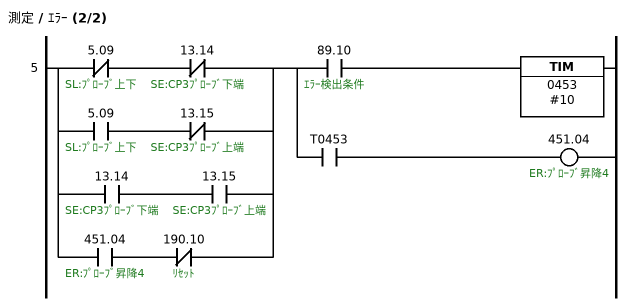
; rung 5
LDNOT 5.09  ; SL:ﾌﾟﾛｰﾌﾞ上下
ANDNOT 13.14  ; SE:CP3ﾌﾟﾛｰﾌﾞ下端
LD 5.09  ; SL:ﾌﾟﾛｰﾌﾞ上下
ANDNOT 13.15  ; SE:CP3ﾌﾟﾛｰﾌﾞ上端
ORLD
LD 13.14  ; SE:CP3ﾌﾟﾛｰﾌﾞ下端
AND 13.15  ; SE:CP3ﾌﾟﾛｰﾌﾞ上端
ORLD
LD 451.04  ; ER:ﾌﾟﾛｰﾌﾞ昇降4
ANDNOT 190.10  ; ﾘｾｯﾄ
ORLD
OUT TR0
AND 89.10  ; ｴﾗｰ検出条件
TIM 0453 #10
LD TR0
AND T0453
OUT 451.04  ; ER:ﾌﾟﾛｰﾌﾞ昇降4

### Section END
; rung 0
END(001)

## Program OV_RV (cyclic task 5)

### Section 制御

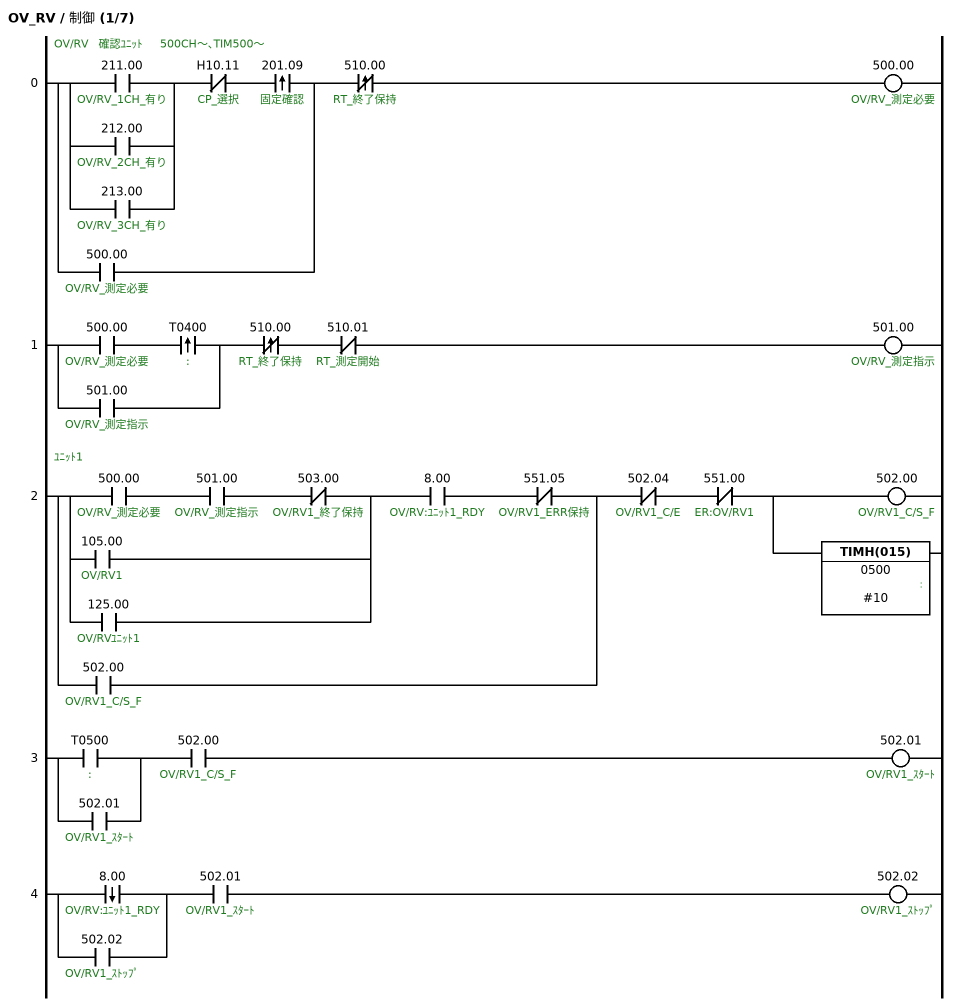
; rung 0: OV/RV   確認ﾕﾆｯﾄ     500CH～､TIM500～
LD 211.00  ; OV/RV_1CH_有り
OR 212.00  ; OV/RV_2CH_有り
OR 213.00  ; OV/RV_3CH_有り
ANDNOT H10.11  ; CP_選択
@AND 201.09  ; 固定確認
OR 500.00  ; OV/RV_測定必要
@ANDNOT 510.00  ; RT_終了保持
OUT 500.00  ; OV/RV_測定必要
; rung 1
LD 500.00  ; OV/RV_測定必要
@AND T0400  ; :
OR 501.00  ; OV/RV_測定指示
@ANDNOT 510.00  ; RT_終了保持
ANDNOT 510.01  ; RT_測定開始
OUT 501.00  ; OV/RV_測定指示
; rung 2: ﾕﾆｯﾄ1
LD 500.00  ; OV/RV_測定必要
AND 501.00  ; OV/RV_測定指示
ANDNOT 503.00  ; OV/RV1_終了保持
OR 105.00  ; OV/RV1
OR 125.00  ; OV/RVﾕﾆｯﾄ1
AND 8.00  ; OV/RV:ﾕﾆｯﾄ1_RDY
ANDNOT 551.05  ; OV/RV1_ERR保持
OR 502.00  ; OV/RV1_C/S_F
ANDNOT 502.04  ; OV/RV1_C/E
ANDNOT 551.00  ; ER:OV/RV1
OUT 502.00  ; OV/RV1_C/S_F
TIMH(015) 0500 #10  ; :
; rung 3
LD T0500  ; :
OR 502.01  ; OV/RV1_ｽﾀｰﾄ
AND 502.00  ; OV/RV1_C/S_F
OUT 502.01  ; OV/RV1_ｽﾀｰﾄ
; rung 4
%LD 8.00  ; OV/RV:ﾕﾆｯﾄ1_RDY
OR 502.02  ; OV/RV1_ｽﾄｯﾌﾟ
AND 502.01  ; OV/RV1_ｽﾀｰﾄ
OUT 502.02  ; OV/RV1_ｽﾄｯﾌﾟ

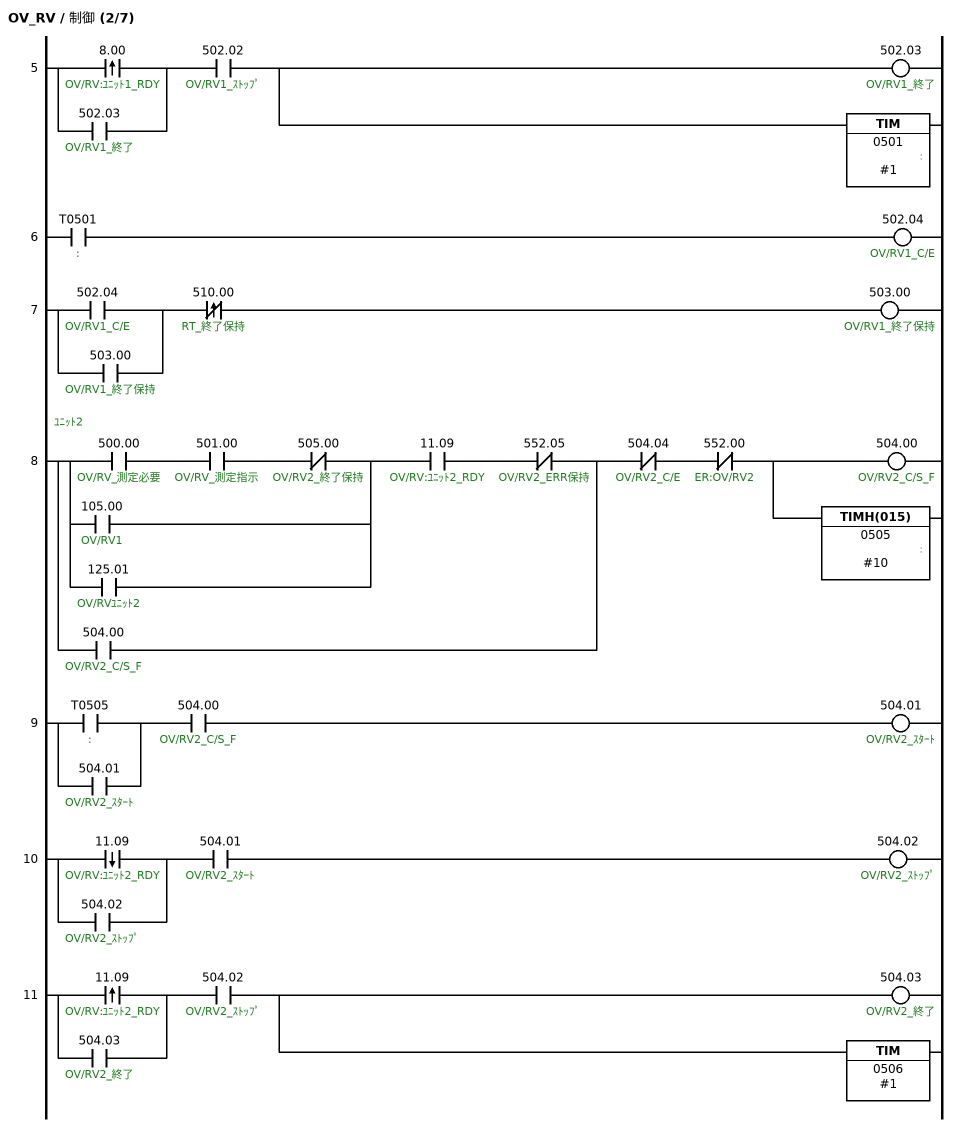
; rung 5
@LD 8.00  ; OV/RV:ﾕﾆｯﾄ1_RDY
OR 502.03  ; OV/RV1_終了
AND 502.02  ; OV/RV1_ｽﾄｯﾌﾟ
OUT 502.03  ; OV/RV1_終了
TIM 0501 #1  ; :
; rung 6
LD T0501  ; :
OUT 502.04  ; OV/RV1_C/E
; rung 7
LD 502.04  ; OV/RV1_C/E
OR 503.00  ; OV/RV1_終了保持
@ANDNOT 510.00  ; RT_終了保持
OUT 503.00  ; OV/RV1_終了保持
; rung 8: ﾕﾆｯﾄ2
LD 500.00  ; OV/RV_測定必要
AND 501.00  ; OV/RV_測定指示
ANDNOT 505.00  ; OV/RV2_終了保持
OR 105.00  ; OV/RV1
OR 125.01  ; OV/RVﾕﾆｯﾄ2
AND 11.09  ; OV/RV:ﾕﾆｯﾄ2_RDY
ANDNOT 552.05  ; OV/RV2_ERR保持
OR 504.00  ; OV/RV2_C/S_F
ANDNOT 504.04  ; OV/RV2_C/E
ANDNOT 552.00  ; ER:OV/RV2
OUT 504.00  ; OV/RV2_C/S_F
TIMH(015) 0505 #10  ; :
; rung 9
LD T0505  ; :
OR 504.01  ; OV/RV2_ｽﾀｰﾄ
AND 504.00  ; OV/RV2_C/S_F
OUT 504.01  ; OV/RV2_ｽﾀｰﾄ
; rung 10
%LD 11.09  ; OV/RV:ﾕﾆｯﾄ2_RDY
OR 504.02  ; OV/RV2_ｽﾄｯﾌﾟ
AND 504.01  ; OV/RV2_ｽﾀｰﾄ
OUT 504.02  ; OV/RV2_ｽﾄｯﾌﾟ
; rung 11
@LD 11.09  ; OV/RV:ﾕﾆｯﾄ2_RDY
OR 504.03  ; OV/RV2_終了
AND 504.02  ; OV/RV2_ｽﾄｯﾌﾟ
OUT 504.03  ; OV/RV2_終了
TIM 0506 #1

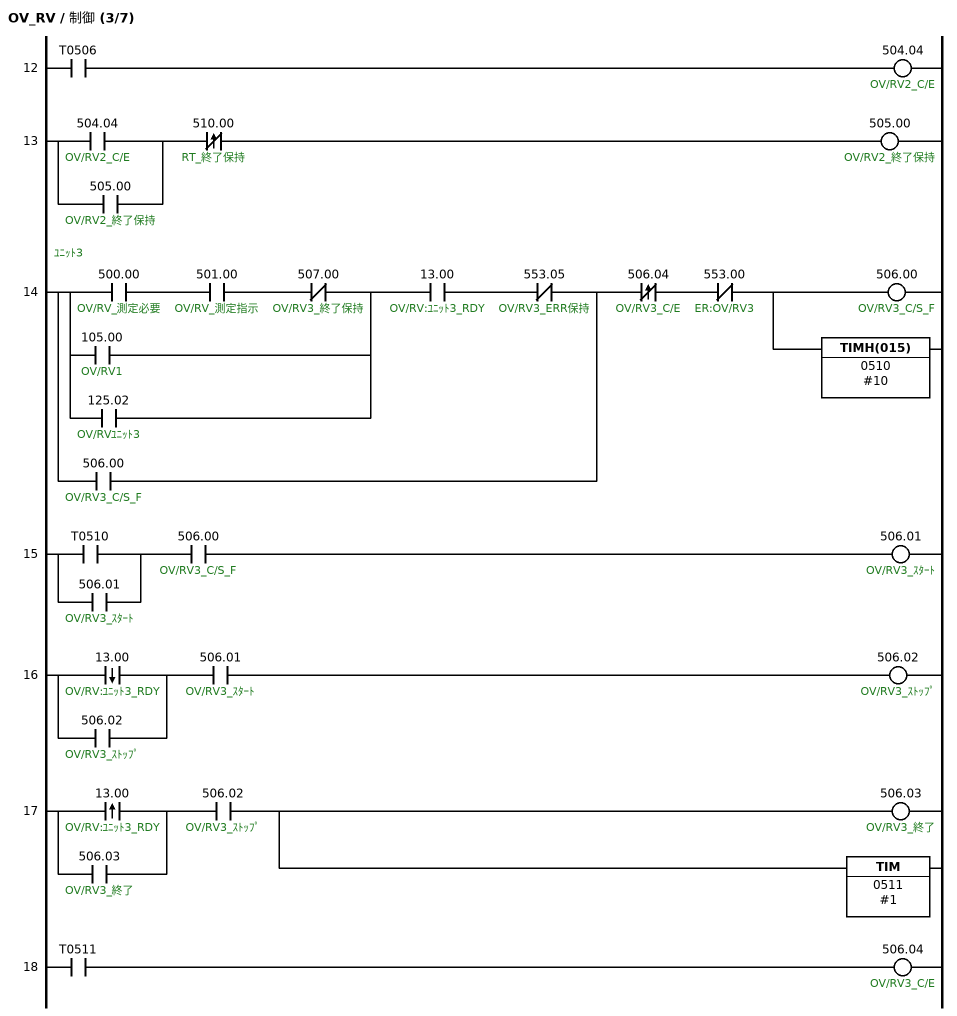
; rung 12
LD T0506
OUT 504.04  ; OV/RV2_C/E
; rung 13
LD 504.04  ; OV/RV2_C/E
OR 505.00  ; OV/RV2_終了保持
@ANDNOT 510.00  ; RT_終了保持
OUT 505.00  ; OV/RV2_終了保持
; rung 14: ﾕﾆｯﾄ3
LD 500.00  ; OV/RV_測定必要
AND 501.00  ; OV/RV_測定指示
ANDNOT 507.00  ; OV/RV3_終了保持
OR 105.00  ; OV/RV1
OR 125.02  ; OV/RVﾕﾆｯﾄ3
AND 13.00  ; OV/RV:ﾕﾆｯﾄ3_RDY
ANDNOT 553.05  ; OV/RV3_ERR保持
OR 506.00  ; OV/RV3_C/S_F
@ANDNOT 506.04  ; OV/RV3_C/E
ANDNOT 553.00  ; ER:OV/RV3
OUT 506.00  ; OV/RV3_C/S_F
TIMH(015) 0510 #10
; rung 15
LD T0510
OR 506.01  ; OV/RV3_ｽﾀｰﾄ
AND 506.00  ; OV/RV3_C/S_F
OUT 506.01  ; OV/RV3_ｽﾀｰﾄ
; rung 16
%LD 13.00  ; OV/RV:ﾕﾆｯﾄ3_RDY
OR 506.02  ; OV/RV3_ｽﾄｯﾌﾟ
AND 506.01  ; OV/RV3_ｽﾀｰﾄ
OUT 506.02  ; OV/RV3_ｽﾄｯﾌﾟ
; rung 17
@LD 13.00  ; OV/RV:ﾕﾆｯﾄ3_RDY
OR 506.03  ; OV/RV3_終了
AND 506.02  ; OV/RV3_ｽﾄｯﾌﾟ
OUT 506.03  ; OV/RV3_終了
TIM 0511 #1
; rung 18
LD T0511
OUT 506.04  ; OV/RV3_C/E

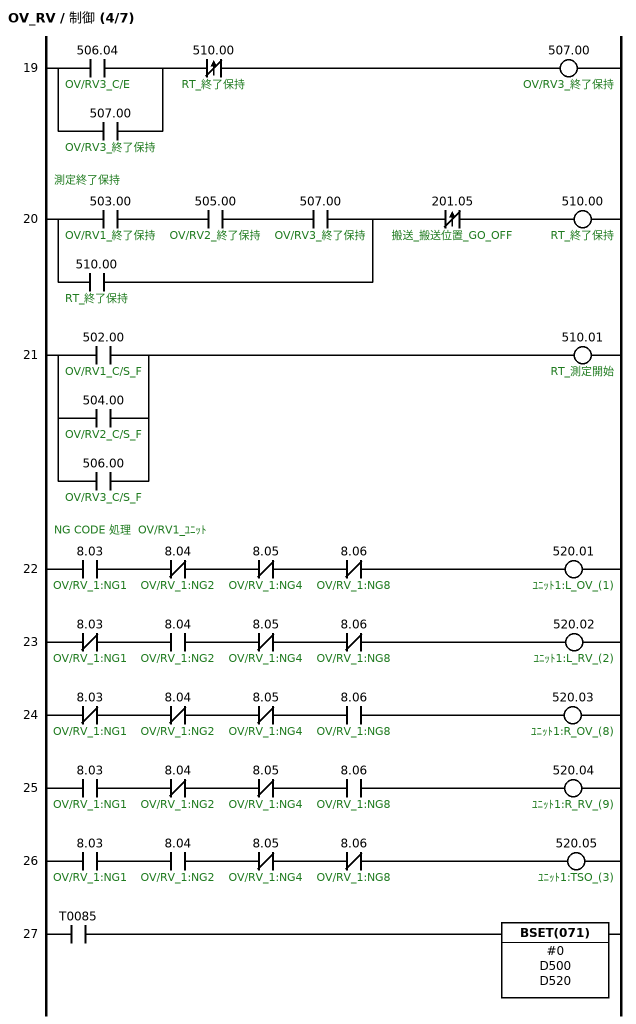
; rung 19
LD 506.04  ; OV/RV3_C/E
OR 507.00  ; OV/RV3_終了保持
@ANDNOT 510.00  ; RT_終了保持
OUT 507.00  ; OV/RV3_終了保持
; rung 20: 測定終了保持
LD 503.00  ; OV/RV1_終了保持
AND 505.00  ; OV/RV2_終了保持
AND 507.00  ; OV/RV3_終了保持
OR 510.00  ; RT_終了保持
@ANDNOT 201.05  ; 搬送_搬送位置_GO_OFF
OUT 510.00  ; RT_終了保持
; rung 21
LD 502.00  ; OV/RV1_C/S_F
OR 504.00  ; OV/RV2_C/S_F
OR 506.00  ; OV/RV3_C/S_F
OUT 510.01  ; RT_測定開始
; rung 22: NG CODE 処理  OV/RV1_ﾕﾆｯﾄ
LD 8.03  ; OV/RV_1:NG1
ANDNOT 8.04  ; OV/RV_1:NG2
ANDNOT 8.05  ; OV/RV_1:NG4
ANDNOT 8.06  ; OV/RV_1:NG8
OUT 520.01  ; ﾕﾆｯﾄ1:L_OV_(1)
; rung 23
LDNOT 8.03  ; OV/RV_1:NG1
AND 8.04  ; OV/RV_1:NG2
ANDNOT 8.05  ; OV/RV_1:NG4
ANDNOT 8.06  ; OV/RV_1:NG8
OUT 520.02  ; ﾕﾆｯﾄ1:L_RV_(2)
; rung 24
LDNOT 8.03  ; OV/RV_1:NG1
ANDNOT 8.04  ; OV/RV_1:NG2
ANDNOT 8.05  ; OV/RV_1:NG4
AND 8.06  ; OV/RV_1:NG8
OUT 520.03  ; ﾕﾆｯﾄ1:R_OV_(8)
; rung 25
LD 8.03  ; OV/RV_1:NG1
ANDNOT 8.04  ; OV/RV_1:NG2
ANDNOT 8.05  ; OV/RV_1:NG4
AND 8.06  ; OV/RV_1:NG8
OUT 520.04  ; ﾕﾆｯﾄ1:R_RV_(9)
; rung 26
LD 8.03  ; OV/RV_1:NG1
AND 8.04  ; OV/RV_1:NG2
ANDNOT 8.05  ; OV/RV_1:NG4
ANDNOT 8.06  ; OV/RV_1:NG8
OUT 520.05  ; ﾕﾆｯﾄ1:TSO_(3)
; rung 27
LD T0085
BSET(071) #0 D500 D520

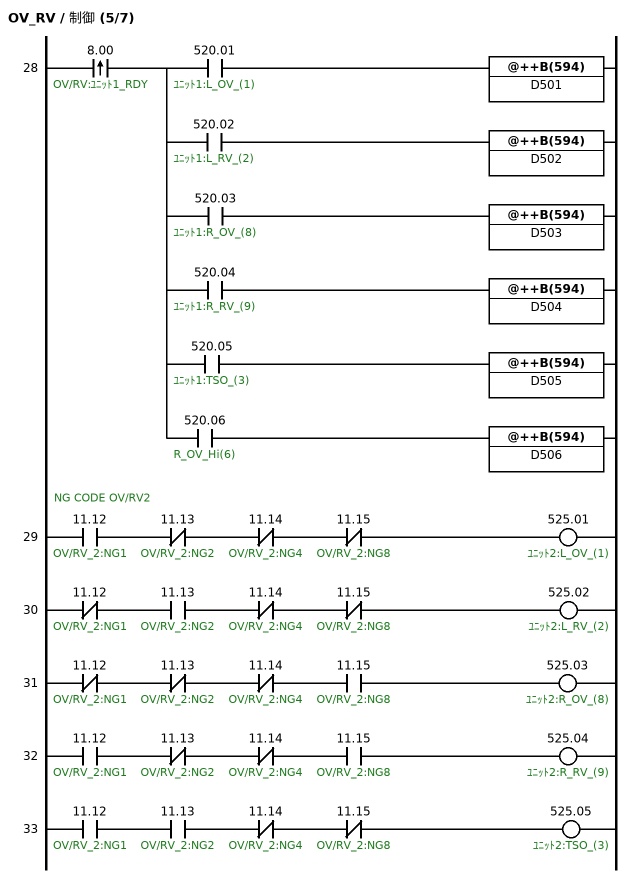
; rung 28
@LD 8.00  ; OV/RV:ﾕﾆｯﾄ1_RDY
OUT TR0
AND 520.01  ; ﾕﾆｯﾄ1:L_OV_(1)
@++B(594) D501
LD TR0
AND 520.02  ; ﾕﾆｯﾄ1:L_RV_(2)
@++B(594) D502
LD TR0
AND 520.03  ; ﾕﾆｯﾄ1:R_OV_(8)
@++B(594) D503
LD TR0
AND 520.04  ; ﾕﾆｯﾄ1:R_RV_(9)
@++B(594) D504
LD TR0
AND 520.05  ; ﾕﾆｯﾄ1:TSO_(3)
@++B(594) D505
LD TR0
AND 520.06  ; R_OV_Hi(6)
@++B(594) D506
; rung 29: NG CODE OV/RV2
LD 11.12  ; OV/RV_2:NG1
ANDNOT 11.13  ; OV/RV_2:NG2
ANDNOT 11.14  ; OV/RV_2:NG4
ANDNOT 11.15  ; OV/RV_2:NG8
OUT 525.01  ; ﾕﾆｯﾄ2:L_OV_(1)
; rung 30
LDNOT 11.12  ; OV/RV_2:NG1
AND 11.13  ; OV/RV_2:NG2
ANDNOT 11.14  ; OV/RV_2:NG4
ANDNOT 11.15  ; OV/RV_2:NG8
OUT 525.02  ; ﾕﾆｯﾄ2:L_RV_(2)
; rung 31
LDNOT 11.12  ; OV/RV_2:NG1
ANDNOT 11.13  ; OV/RV_2:NG2
ANDNOT 11.14  ; OV/RV_2:NG4
AND 11.15  ; OV/RV_2:NG8
OUT 525.03  ; ﾕﾆｯﾄ2:R_OV_(8)
; rung 32
LD 11.12  ; OV/RV_2:NG1
ANDNOT 11.13  ; OV/RV_2:NG2
ANDNOT 11.14  ; OV/RV_2:NG4
AND 11.15  ; OV/RV_2:NG8
OUT 525.04  ; ﾕﾆｯﾄ2:R_RV_(9)
; rung 33
LD 11.12  ; OV/RV_2:NG1
AND 11.13  ; OV/RV_2:NG2
ANDNOT 11.14  ; OV/RV_2:NG4
ANDNOT 11.15  ; OV/RV_2:NG8
OUT 525.05  ; ﾕﾆｯﾄ2:TSO_(3)

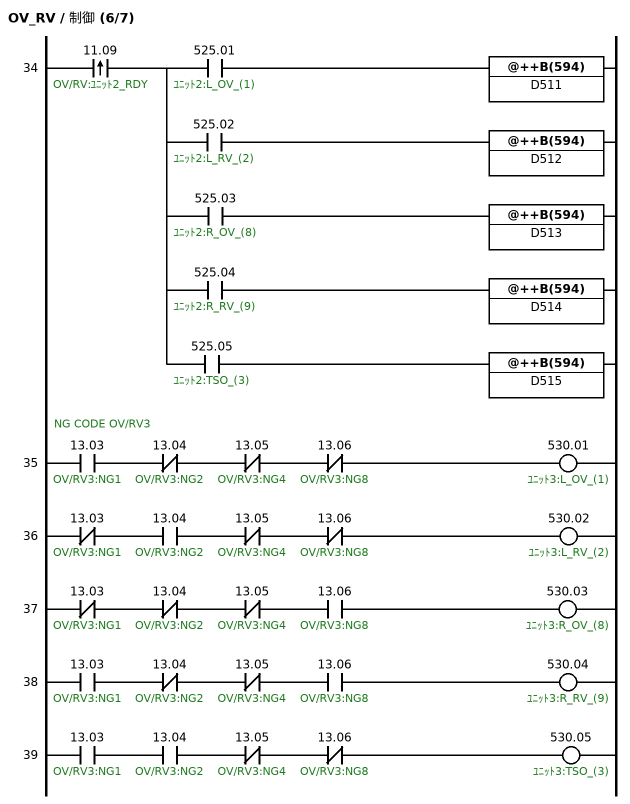
; rung 34
@LD 11.09  ; OV/RV:ﾕﾆｯﾄ2_RDY
OUT TR0
AND 525.01  ; ﾕﾆｯﾄ2:L_OV_(1)
@++B(594) D511
LD TR0
AND 525.02  ; ﾕﾆｯﾄ2:L_RV_(2)
@++B(594) D512
LD TR0
AND 525.03  ; ﾕﾆｯﾄ2:R_OV_(8)
@++B(594) D513
LD TR0
AND 525.04  ; ﾕﾆｯﾄ2:R_RV_(9)
@++B(594) D514
LD TR0
AND 525.05  ; ﾕﾆｯﾄ2:TSO_(3)
@++B(594) D515
; rung 35: NG CODE OV/RV3
LD 13.03  ; OV/RV3:NG1
ANDNOT 13.04  ; OV/RV3:NG2
ANDNOT 13.05  ; OV/RV3:NG4
ANDNOT 13.06  ; OV/RV3:NG8
OUT 530.01  ; ﾕﾆｯﾄ3:L_OV_(1)
; rung 36
LDNOT 13.03  ; OV/RV3:NG1
AND 13.04  ; OV/RV3:NG2
ANDNOT 13.05  ; OV/RV3:NG4
ANDNOT 13.06  ; OV/RV3:NG8
OUT 530.02  ; ﾕﾆｯﾄ3:L_RV_(2)
; rung 37
LDNOT 13.03  ; OV/RV3:NG1
ANDNOT 13.04  ; OV/RV3:NG2
ANDNOT 13.05  ; OV/RV3:NG4
AND 13.06  ; OV/RV3:NG8
OUT 530.03  ; ﾕﾆｯﾄ3:R_OV_(8)
; rung 38
LD 13.03  ; OV/RV3:NG1
ANDNOT 13.04  ; OV/RV3:NG2
ANDNOT 13.05  ; OV/RV3:NG4
AND 13.06  ; OV/RV3:NG8
OUT 530.04  ; ﾕﾆｯﾄ3:R_RV_(9)
; rung 39
LD 13.03  ; OV/RV3:NG1
AND 13.04  ; OV/RV3:NG2
ANDNOT 13.05  ; OV/RV3:NG4
ANDNOT 13.06  ; OV/RV3:NG8
OUT 530.05  ; ﾕﾆｯﾄ3:TSO_(3)

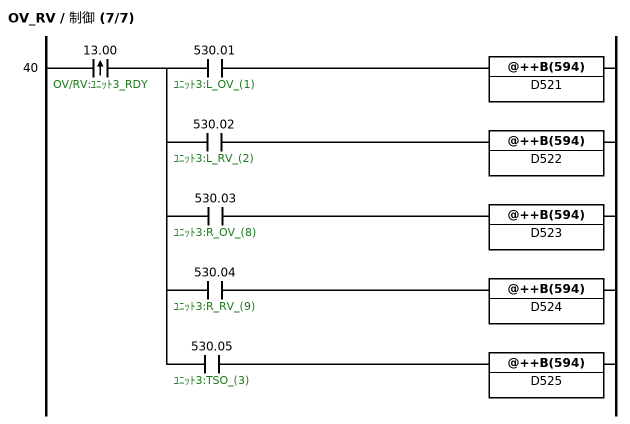
; rung 40
@LD 13.00  ; OV/RV:ﾕﾆｯﾄ3_RDY
OUT TR0
AND 530.01  ; ﾕﾆｯﾄ3:L_OV_(1)
@++B(594) D521
LD TR0
AND 530.02  ; ﾕﾆｯﾄ3:L_RV_(2)
@++B(594) D522
LD TR0
AND 530.03  ; ﾕﾆｯﾄ3:R_OV_(8)
@++B(594) D523
LD TR0
AND 530.04  ; ﾕﾆｯﾄ3:R_RV_(9)
@++B(594) D524
LD TR0
AND 530.05  ; ﾕﾆｯﾄ3:TSO_(3)
@++B(594) D525

### Section 出力
; rung 0: 出力

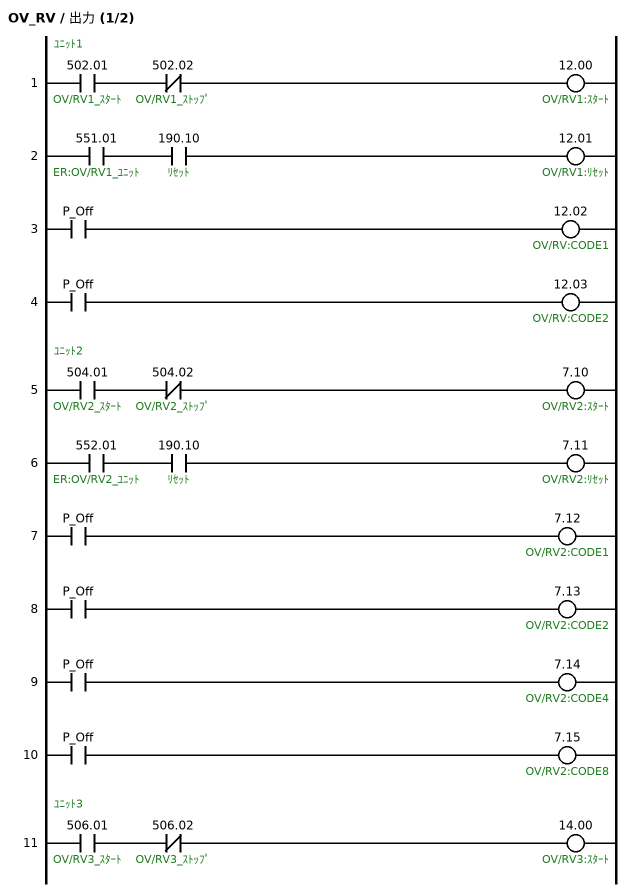
; rung 1: ﾕﾆｯﾄ1
LD 502.01  ; OV/RV1_ｽﾀｰﾄ
ANDNOT 502.02  ; OV/RV1_ｽﾄｯﾌﾟ
OUT 12.00  ; OV/RV1:ｽﾀｰﾄ
; rung 2
LD 551.01  ; ER:OV/RV1_ﾕﾆｯﾄ
AND 190.10  ; ﾘｾｯﾄ
OUT 12.01  ; OV/RV1:ﾘｾｯﾄ
; rung 3
LD P_Off
OUT 12.02  ; OV/RV:CODE1
; rung 4
LD P_Off
OUT 12.03  ; OV/RV:CODE2
; rung 5: ﾕﾆｯﾄ2
LD 504.01  ; OV/RV2_ｽﾀｰﾄ
ANDNOT 504.02  ; OV/RV2_ｽﾄｯﾌﾟ
OUT 7.10  ; OV/RV2:ｽﾀｰﾄ
; rung 6
LD 552.01  ; ER:OV/RV2_ﾕﾆｯﾄ
AND 190.10  ; ﾘｾｯﾄ
OUT 7.11  ; OV/RV2:ﾘｾｯﾄ
; rung 7
LD P_Off
OUT 7.12  ; OV/RV2:CODE1
; rung 8
LD P_Off
OUT 7.13  ; OV/RV2:CODE2
; rung 9
LD P_Off
OUT 7.14  ; OV/RV2:CODE4
; rung 10
LD P_Off
OUT 7.15  ; OV/RV2:CODE8
; rung 11: ﾕﾆｯﾄ3
LD 506.01  ; OV/RV3_ｽﾀｰﾄ
ANDNOT 506.02  ; OV/RV3_ｽﾄｯﾌﾟ
OUT 14.00  ; OV/RV3:ｽﾀｰﾄ

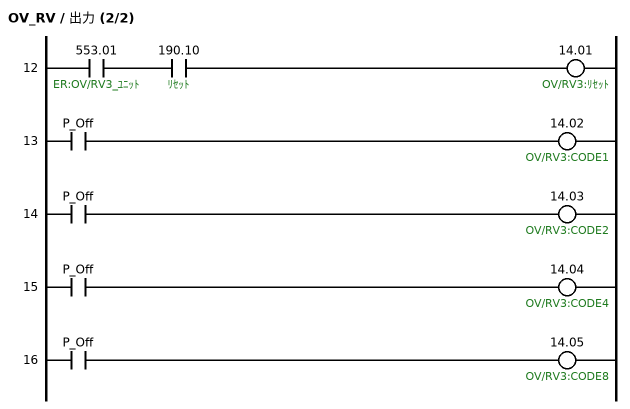
; rung 12
LD 553.01  ; ER:OV/RV3_ﾕﾆｯﾄ
AND 190.10  ; ﾘｾｯﾄ
OUT 14.01  ; OV/RV3:ﾘｾｯﾄ
; rung 13
LD P_Off
OUT 14.02  ; OV/RV3:CODE1
; rung 14
LD P_Off
OUT 14.03  ; OV/RV3:CODE2
; rung 15
LD P_Off
OUT 14.04  ; OV/RV3:CODE4
; rung 16
LD P_Off
OUT 14.05  ; OV/RV3:CODE8

### Section ｴﾗｰ

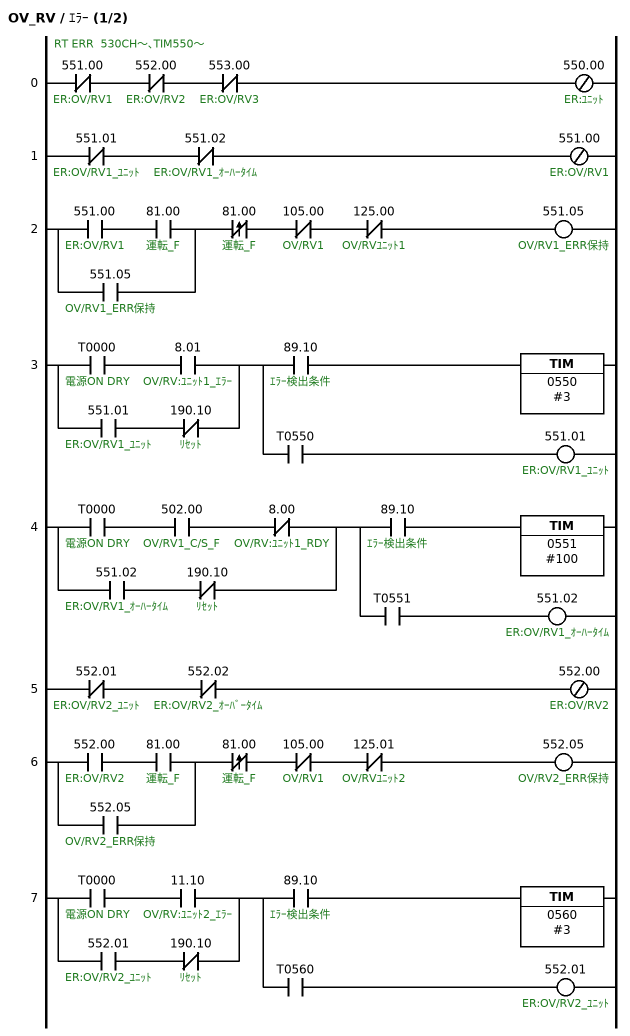
; rung 0: RT ERR  530CH～､TIM550～
LDNOT 551.00  ; ER:OV/RV1
ANDNOT 552.00  ; ER:OV/RV2
ANDNOT 553.00  ; ER:OV/RV3
OUTNOT 550.00  ; ER:ﾕﾆｯﾄ
; rung 1
LDNOT 551.01  ; ER:OV/RV1_ﾕﾆｯﾄ
ANDNOT 551.02  ; ER:OV/RV1_ｵｰﾊｰﾀｲﾑ
OUTNOT 551.00  ; ER:OV/RV1
; rung 2
LD 551.00  ; ER:OV/RV1
AND 81.00  ; 運転_F
OR 551.05  ; OV/RV1_ERR保持
@ANDNOT 81.00  ; 運転_F
ANDNOT 105.00  ; OV/RV1
ANDNOT 125.00  ; OV/RVﾕﾆｯﾄ1
OUT 551.05  ; OV/RV1_ERR保持
; rung 3
LD T0000  ; 電源ON DRY
AND 8.01  ; OV/RV:ﾕﾆｯﾄ1_ｴﾗｰ
LD 551.01  ; ER:OV/RV1_ﾕﾆｯﾄ
ANDNOT 190.10  ; ﾘｾｯﾄ
ORLD
OUT TR0
AND 89.10  ; ｴﾗｰ検出条件
TIM 0550 #3
LD TR0
AND T0550
OUT 551.01  ; ER:OV/RV1_ﾕﾆｯﾄ
; rung 4
LD T0000  ; 電源ON DRY
AND 502.00  ; OV/RV1_C/S_F
ANDNOT 8.00  ; OV/RV:ﾕﾆｯﾄ1_RDY
LD 551.02  ; ER:OV/RV1_ｵｰﾊｰﾀｲﾑ
ANDNOT 190.10  ; ﾘｾｯﾄ
ORLD
OUT TR0
AND 89.10  ; ｴﾗｰ検出条件
TIM 0551 #100
LD TR0
AND T0551
OUT 551.02  ; ER:OV/RV1_ｵｰﾊｰﾀｲﾑ
; rung 5
LDNOT 552.01  ; ER:OV/RV2_ﾕﾆｯﾄ
ANDNOT 552.02  ; ER:OV/RV2_ｵｰﾊﾞｰﾀｲﾑ
OUTNOT 552.00  ; ER:OV/RV2
; rung 6
LD 552.00  ; ER:OV/RV2
AND 81.00  ; 運転_F
OR 552.05  ; OV/RV2_ERR保持
@ANDNOT 81.00  ; 運転_F
ANDNOT 105.00  ; OV/RV1
ANDNOT 125.01  ; OV/RVﾕﾆｯﾄ2
OUT 552.05  ; OV/RV2_ERR保持
; rung 7
LD T0000  ; 電源ON DRY
AND 11.10  ; OV/RV:ﾕﾆｯﾄ2_ｴﾗｰ
LD 552.01  ; ER:OV/RV2_ﾕﾆｯﾄ
ANDNOT 190.10  ; ﾘｾｯﾄ
ORLD
OUT TR0
AND 89.10  ; ｴﾗｰ検出条件
TIM 0560 #3
LD TR0
AND T0560
OUT 552.01  ; ER:OV/RV2_ﾕﾆｯﾄ

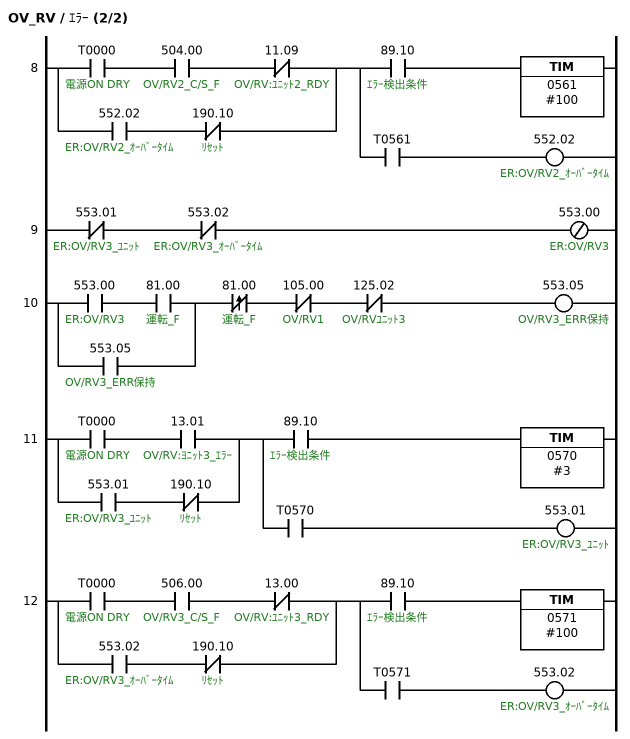
; rung 8
LD T0000  ; 電源ON DRY
AND 504.00  ; OV/RV2_C/S_F
ANDNOT 11.09  ; OV/RV:ﾕﾆｯﾄ2_RDY
LD 552.02  ; ER:OV/RV2_ｵｰﾊﾞｰﾀｲﾑ
ANDNOT 190.10  ; ﾘｾｯﾄ
ORLD
OUT TR0
AND 89.10  ; ｴﾗｰ検出条件
TIM 0561 #100
LD TR0
AND T0561
OUT 552.02  ; ER:OV/RV2_ｵｰﾊﾞｰﾀｲﾑ
; rung 9
LDNOT 553.01  ; ER:OV/RV3_ﾕﾆｯﾄ
ANDNOT 553.02  ; ER:OV/RV3_ｵｰﾊﾞｰﾀｲﾑ
OUTNOT 553.00  ; ER:OV/RV3
; rung 10
LD 553.00  ; ER:OV/RV3
AND 81.00  ; 運転_F
OR 553.05  ; OV/RV3_ERR保持
@ANDNOT 81.00  ; 運転_F
ANDNOT 105.00  ; OV/RV1
ANDNOT 125.02  ; OV/RVﾕﾆｯﾄ3
OUT 553.05  ; OV/RV3_ERR保持
; rung 11
LD T0000  ; 電源ON DRY
AND 13.01  ; OV/RV:ﾖﾆｯﾄ3_ｴﾗｰ
LD 553.01  ; ER:OV/RV3_ﾕﾆｯﾄ
ANDNOT 190.10  ; ﾘｾｯﾄ
ORLD
OUT TR0
AND 89.10  ; ｴﾗｰ検出条件
TIM 0570 #3
LD TR0
AND T0570
OUT 553.01  ; ER:OV/RV3_ﾕﾆｯﾄ
; rung 12
LD T0000  ; 電源ON DRY
AND 506.00  ; OV/RV3_C/S_F
ANDNOT 13.00  ; OV/RV:ﾕﾆｯﾄ3_RDY
LD 553.02  ; ER:OV/RV3_ｵｰﾊﾞｰﾀｲﾑ
ANDNOT 190.10  ; ﾘｾｯﾄ
ORLD
OUT TR0
AND 89.10  ; ｴﾗｰ検出条件
TIM 0571 #100
LD TR0
AND T0571
OUT 553.02  ; ER:OV/RV3_ｵｰﾊﾞｰﾀｲﾑ

### Section END
; rung 0
END(001)

## Program CP (cyclic task 6)

### Section 制御

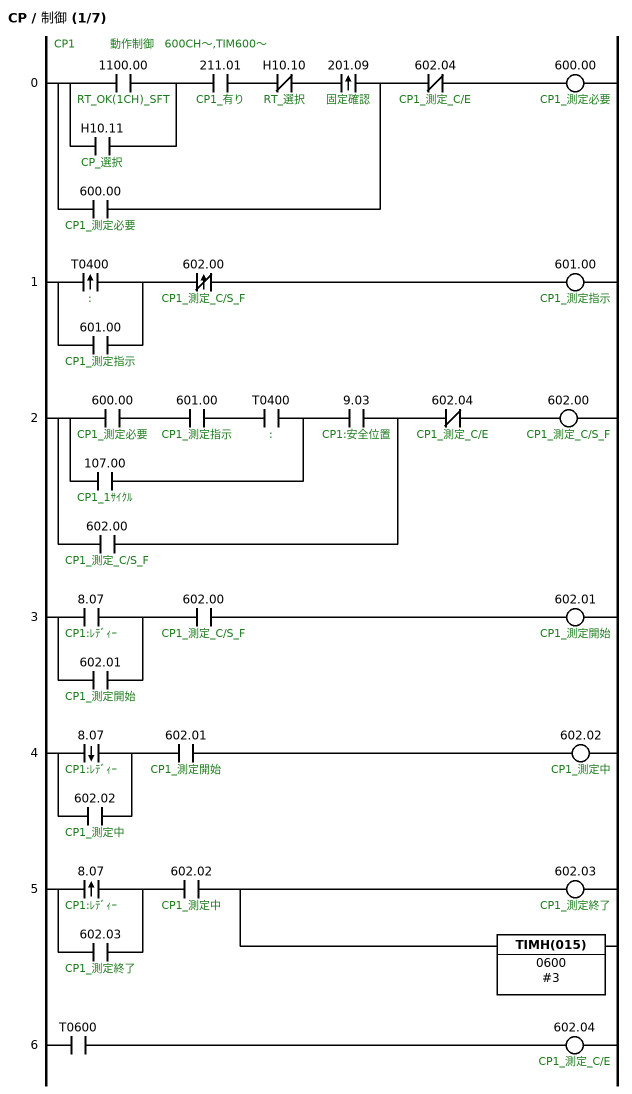
; rung 0: CP1          動作制御   600CH～,TIM600～
LD 1100.00  ; RT_OK(1CH)_SFT
OR H10.11  ; CP_選択
AND 211.01  ; CP1_有り
ANDNOT H10.10  ; RT_選択
@AND 201.09  ; 固定確認
OR 600.00  ; CP1_測定必要
ANDNOT 602.04  ; CP1_測定_C/E
OUT 600.00  ; CP1_測定必要
; rung 1
@LD T0400  ; :
OR 601.00  ; CP1_測定指示
@ANDNOT 602.00  ; CP1_測定_C/S_F
OUT 601.00  ; CP1_測定指示
; rung 2
LD 600.00  ; CP1_測定必要
AND 601.00  ; CP1_測定指示
AND T0400  ; :
OR 107.00  ; CP1_1ｻｲｸﾙ
AND 9.03  ; CP1:安全位置
OR 602.00  ; CP1_測定_C/S_F
ANDNOT 602.04  ; CP1_測定_C/E
OUT 602.00  ; CP1_測定_C/S_F
; rung 3
LD 8.07  ; CP1:ﾚﾃﾞｨｰ
OR 602.01  ; CP1_測定開始
AND 602.00  ; CP1_測定_C/S_F
OUT 602.01  ; CP1_測定開始
; rung 4
%LD 8.07  ; CP1:ﾚﾃﾞｨｰ
OR 602.02  ; CP1_測定中
AND 602.01  ; CP1_測定開始
OUT 602.02  ; CP1_測定中
; rung 5
@LD 8.07  ; CP1:ﾚﾃﾞｨｰ
OR 602.03  ; CP1_測定終了
AND 602.02  ; CP1_測定中
OUT 602.03  ; CP1_測定終了
TIMH(015) 0600 #3
; rung 6
LD T0600
OUT 602.04  ; CP1_測定_C/E

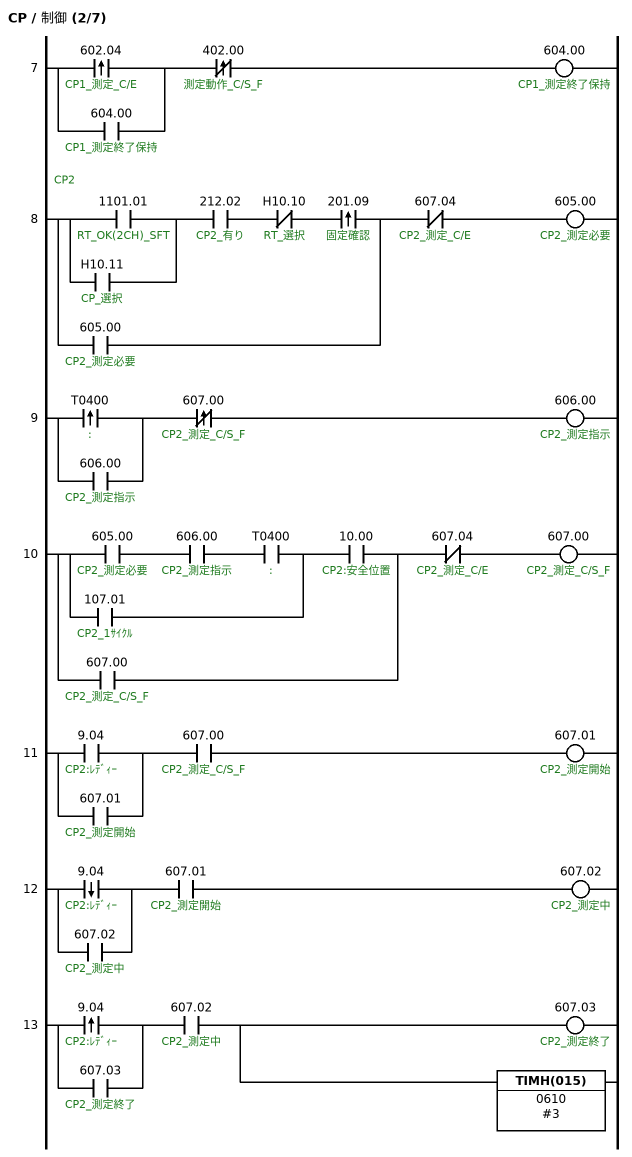
; rung 7
@LD 602.04  ; CP1_測定_C/E
OR 604.00  ; CP1_測定終了保持
@ANDNOT 402.00  ; 測定動作_C/S_F
OUT 604.00  ; CP1_測定終了保持
; rung 8: CP2
LD 1101.01  ; RT_OK(2CH)_SFT
OR H10.11  ; CP_選択
AND 212.02  ; CP2_有り
ANDNOT H10.10  ; RT_選択
@AND 201.09  ; 固定確認
OR 605.00  ; CP2_測定必要
ANDNOT 607.04  ; CP2_測定_C/E
OUT 605.00  ; CP2_測定必要
; rung 9
@LD T0400  ; :
OR 606.00  ; CP2_測定指示
@ANDNOT 607.00  ; CP2_測定_C/S_F
OUT 606.00  ; CP2_測定指示
; rung 10
LD 605.00  ; CP2_測定必要
AND 606.00  ; CP2_測定指示
AND T0400  ; :
OR 107.01  ; CP2_1ｻｲｸﾙ
AND 10.00  ; CP2:安全位置
OR 607.00  ; CP2_測定_C/S_F
ANDNOT 607.04  ; CP2_測定_C/E
OUT 607.00  ; CP2_測定_C/S_F
; rung 11
LD 9.04  ; CP2:ﾚﾃﾞｨｰ
OR 607.01  ; CP2_測定開始
AND 607.00  ; CP2_測定_C/S_F
OUT 607.01  ; CP2_測定開始
; rung 12
%LD 9.04  ; CP2:ﾚﾃﾞｨｰ
OR 607.02  ; CP2_測定中
AND 607.01  ; CP2_測定開始
OUT 607.02  ; CP2_測定中
; rung 13
@LD 9.04  ; CP2:ﾚﾃﾞｨｰ
OR 607.03  ; CP2_測定終了
AND 607.02  ; CP2_測定中
OUT 607.03  ; CP2_測定終了
TIMH(015) 0610 #3

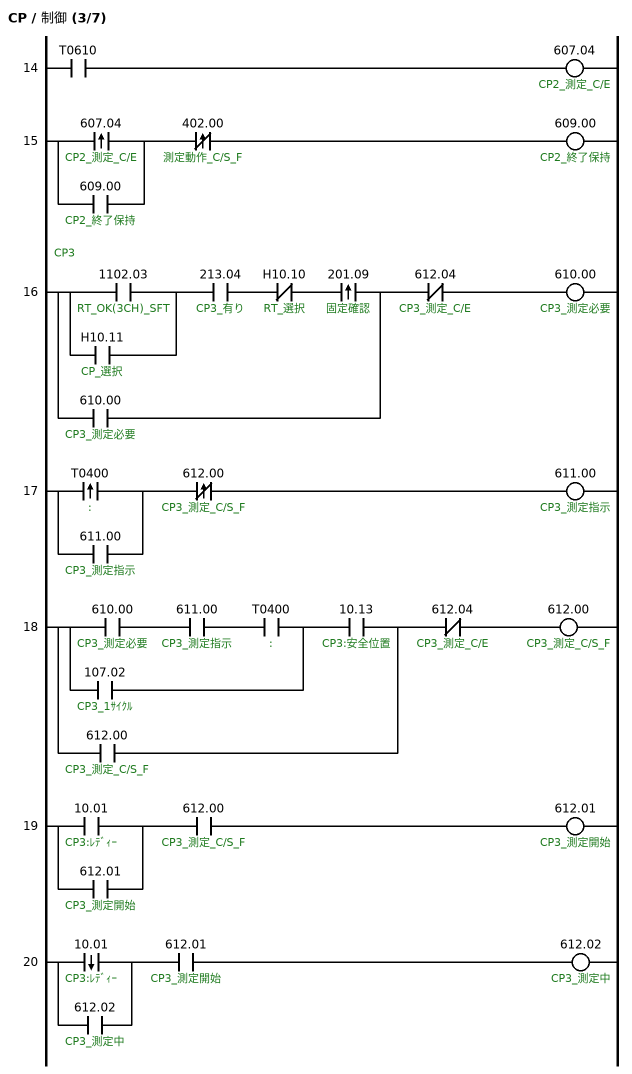
; rung 14
LD T0610
OUT 607.04  ; CP2_測定_C/E
; rung 15
@LD 607.04  ; CP2_測定_C/E
OR 609.00  ; CP2_終了保持
@ANDNOT 402.00  ; 測定動作_C/S_F
OUT 609.00  ; CP2_終了保持
; rung 16: CP3
LD 1102.03  ; RT_OK(3CH)_SFT
OR H10.11  ; CP_選択
AND 213.04  ; CP3_有り
ANDNOT H10.10  ; RT_選択
@AND 201.09  ; 固定確認
OR 610.00  ; CP3_測定必要
ANDNOT 612.04  ; CP3_測定_C/E
OUT 610.00  ; CP3_測定必要
; rung 17
@LD T0400  ; :
OR 611.00  ; CP3_測定指示
@ANDNOT 612.00  ; CP3_測定_C/S_F
OUT 611.00  ; CP3_測定指示
; rung 18
LD 610.00  ; CP3_測定必要
AND 611.00  ; CP3_測定指示
AND T0400  ; :
OR 107.02  ; CP3_1ｻｲｸﾙ
AND 10.13  ; CP3:安全位置
OR 612.00  ; CP3_測定_C/S_F
ANDNOT 612.04  ; CP3_測定_C/E
OUT 612.00  ; CP3_測定_C/S_F
; rung 19
LD 10.01  ; CP3:ﾚﾃﾞｨｰ
OR 612.01  ; CP3_測定開始
AND 612.00  ; CP3_測定_C/S_F
OUT 612.01  ; CP3_測定開始
; rung 20
%LD 10.01  ; CP3:ﾚﾃﾞｨｰ
OR 612.02  ; CP3_測定中
AND 612.01  ; CP3_測定開始
OUT 612.02  ; CP3_測定中

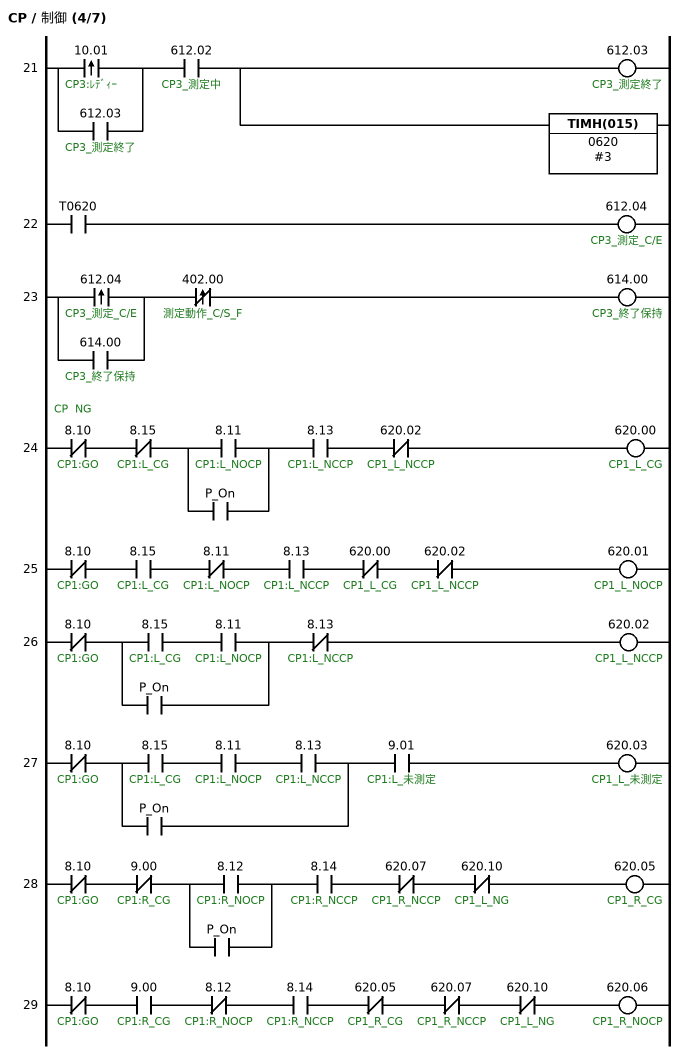
; rung 21
@LD 10.01  ; CP3:ﾚﾃﾞｨｰ
OR 612.03  ; CP3_測定終了
AND 612.02  ; CP3_測定中
OUT 612.03  ; CP3_測定終了
TIMH(015) 0620 #3
; rung 22
LD T0620
OUT 612.04  ; CP3_測定_C/E
; rung 23
@LD 612.04  ; CP3_測定_C/E
OR 614.00  ; CP3_終了保持
@ANDNOT 402.00  ; 測定動作_C/S_F
OUT 614.00  ; CP3_終了保持
; rung 24: CP  NG
LDNOT 8.10  ; CP1:GO
ANDNOT 8.15  ; CP1:L_CG
LD 8.11  ; CP1:L_NOCP
OR P_On  // 2015/11/13変更
ANDLD
AND 8.13  ; CP1:L_NCCP
ANDNOT 620.02  ; CP1_L_NCCP  // 2015/11/13変更
OUT 620.00  ; CP1_L_CG
; rung 25
LDNOT 8.10  ; CP1:GO
AND 8.15  ; CP1:L_CG
ANDNOT 8.11  ; CP1:L_NOCP
AND 8.13  ; CP1:L_NCCP
ANDNOT 620.00  ; CP1_L_CG
ANDNOT 620.02  ; CP1_L_NCCP  // 2015/11/13変更
OUT 620.01  ; CP1_L_NOCP
; rung 26
LDNOT 8.10  ; CP1:GO
LD 8.15  ; CP1:L_CG
AND 8.11  ; CP1:L_NOCP
OR P_On  // 2015/11/13変更
ANDLD
ANDNOT 8.13  ; CP1:L_NCCP
OUT 620.02  ; CP1_L_NCCP
; rung 27
LDNOT 8.10  ; CP1:GO
LD 8.15  ; CP1:L_CG
AND 8.11  ; CP1:L_NOCP
AND 8.13  ; CP1:L_NCCP
OR P_On  // 2015/11/13変更
ANDLD
AND 9.01  ; CP1:L_未測定  // 2015/11/13変更
OUT 620.03  ; CP1_L_未測定
; rung 28
LDNOT 8.10  ; CP1:GO
ANDNOT 9.00  ; CP1:R_CG
LD 8.12  ; CP1:R_NOCP
OR P_On  // 2015/11/13変更
ANDLD
AND 8.14  ; CP1:R_NCCP
ANDNOT 620.07  ; CP1_R_NCCP
ANDNOT 620.10  ; CP1_L_NG
OUT 620.05  ; CP1_R_CG
; rung 29
LDNOT 8.10  ; CP1:GO
AND 9.00  ; CP1:R_CG
ANDNOT 8.12  ; CP1:R_NOCP
AND 8.14  ; CP1:R_NCCP
ANDNOT 620.05  ; CP1_R_CG
ANDNOT 620.07  ; CP1_R_NCCP
ANDNOT 620.10  ; CP1_L_NG
OUT 620.06  ; CP1_R_NOCP

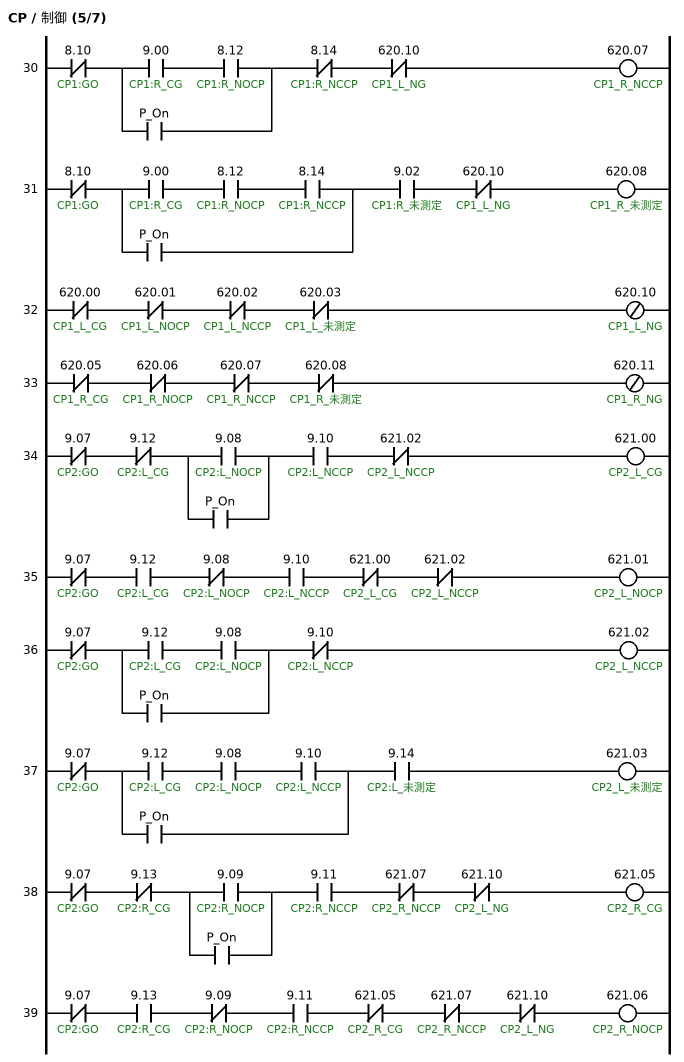
; rung 30
LDNOT 8.10  ; CP1:GO
LD 9.00  ; CP1:R_CG
AND 8.12  ; CP1:R_NOCP
OR P_On  // 2015/11/13変更
ANDLD
ANDNOT 8.14  ; CP1:R_NCCP
ANDNOT 620.10  ; CP1_L_NG
OUT 620.07  ; CP1_R_NCCP
; rung 31
LDNOT 8.10  ; CP1:GO
LD 9.00  ; CP1:R_CG
AND 8.12  ; CP1:R_NOCP
AND 8.14  ; CP1:R_NCCP
OR P_On  // 2015/11/13変更
ANDLD
AND 9.02  ; CP1:R_未測定  // 2015/11/13変更
ANDNOT 620.10  ; CP1_L_NG
OUT 620.08  ; CP1_R_未測定
; rung 32
LDNOT 620.00  ; CP1_L_CG
ANDNOT 620.01  ; CP1_L_NOCP
ANDNOT 620.02  ; CP1_L_NCCP
ANDNOT 620.03  ; CP1_L_未測定
OUTNOT 620.10  ; CP1_L_NG
; rung 33
LDNOT 620.05  ; CP1_R_CG
ANDNOT 620.06  ; CP1_R_NOCP
ANDNOT 620.07  ; CP1_R_NCCP
ANDNOT 620.08  ; CP1_R_未測定
OUTNOT 620.11  ; CP1_R_NG
; rung 34
LDNOT 9.07  ; CP2:GO
ANDNOT 9.12  ; CP2:L_CG
LD 9.08  ; CP2:L_NOCP
OR P_On  // 2015/11/13変更
ANDLD
AND 9.10  ; CP2:L_NCCP
ANDNOT 621.02  ; CP2_L_NCCP
OUT 621.00  ; CP2_L_CG
; rung 35
LDNOT 9.07  ; CP2:GO
AND 9.12  ; CP2:L_CG
ANDNOT 9.08  ; CP2:L_NOCP
AND 9.10  ; CP2:L_NCCP
ANDNOT 621.00  ; CP2_L_CG
ANDNOT 621.02  ; CP2_L_NCCP
OUT 621.01  ; CP2_L_NOCP
; rung 36
LDNOT 9.07  ; CP2:GO
LD 9.12  ; CP2:L_CG
AND 9.08  ; CP2:L_NOCP
OR P_On  // 2015/11/13変更
ANDLD
ANDNOT 9.10  ; CP2:L_NCCP
OUT 621.02  ; CP2_L_NCCP
; rung 37
LDNOT 9.07  ; CP2:GO
LD 9.12  ; CP2:L_CG
AND 9.08  ; CP2:L_NOCP
AND 9.10  ; CP2:L_NCCP
OR P_On  // 2015/11/13変更
ANDLD
AND 9.14  ; CP2:L_未測定  // 2015/11/13変更
OUT 621.03  ; CP2_L_未測定
; rung 38
LDNOT 9.07  ; CP2:GO
ANDNOT 9.13  ; CP2:R_CG
LD 9.09  ; CP2:R_NOCP
OR P_On  // 2015/11/13変更
ANDLD
AND 9.11  ; CP2:R_NCCP
ANDNOT 621.07  ; CP2_R_NCCP
ANDNOT 621.10  ; CP2_L_NG
OUT 621.05  ; CP2_R_CG
; rung 39
LDNOT 9.07  ; CP2:GO
AND 9.13  ; CP2:R_CG
ANDNOT 9.09  ; CP2:R_NOCP
AND 9.11  ; CP2:R_NCCP
ANDNOT 621.05  ; CP2_R_CG
ANDNOT 621.07  ; CP2_R_NCCP
ANDNOT 621.10  ; CP2_L_NG
OUT 621.06  ; CP2_R_NOCP

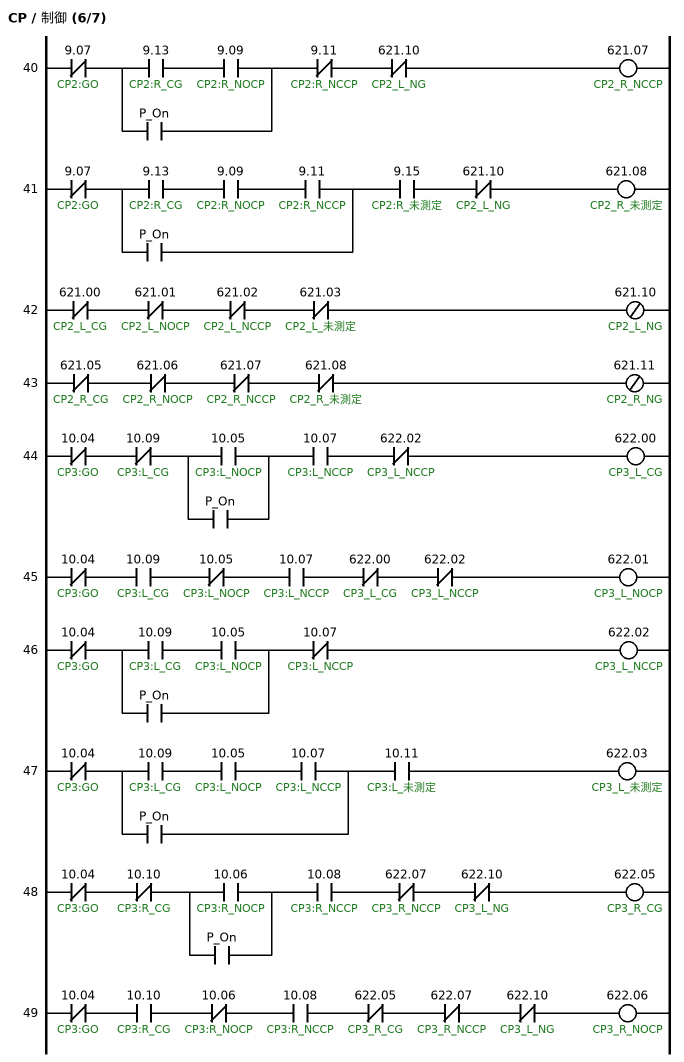
; rung 40
LDNOT 9.07  ; CP2:GO
LD 9.13  ; CP2:R_CG
AND 9.09  ; CP2:R_NOCP
OR P_On  // 2015/11/13変更
ANDLD
ANDNOT 9.11  ; CP2:R_NCCP
ANDNOT 621.10  ; CP2_L_NG
OUT 621.07  ; CP2_R_NCCP
; rung 41
LDNOT 9.07  ; CP2:GO
LD 9.13  ; CP2:R_CG
AND 9.09  ; CP2:R_NOCP
AND 9.11  ; CP2:R_NCCP
OR P_On  // 2015/11/13変更
ANDLD
AND 9.15  ; CP2:R_未測定  // 2015/11/13変更
ANDNOT 621.10  ; CP2_L_NG
OUT 621.08  ; CP2_R_未測定
; rung 42
LDNOT 621.00  ; CP2_L_CG
ANDNOT 621.01  ; CP2_L_NOCP
ANDNOT 621.02  ; CP2_L_NCCP
ANDNOT 621.03  ; CP2_L_未測定
OUTNOT 621.10  ; CP2_L_NG
; rung 43
LDNOT 621.05  ; CP2_R_CG
ANDNOT 621.06  ; CP2_R_NOCP
ANDNOT 621.07  ; CP2_R_NCCP
ANDNOT 621.08  ; CP2_R_未測定
OUTNOT 621.11  ; CP2_R_NG
; rung 44
LDNOT 10.04  ; CP3:GO
ANDNOT 10.09  ; CP3:L_CG
LD 10.05  ; CP3:L_NOCP
OR P_On  // 2015/11/13変更
ANDLD
AND 10.07  ; CP3:L_NCCP
ANDNOT 622.02  ; CP3_L_NCCP
OUT 622.00  ; CP3_L_CG
; rung 45
LDNOT 10.04  ; CP3:GO
AND 10.09  ; CP3:L_CG
ANDNOT 10.05  ; CP3:L_NOCP
AND 10.07  ; CP3:L_NCCP
ANDNOT 622.00  ; CP3_L_CG
ANDNOT 622.02  ; CP3_L_NCCP
OUT 622.01  ; CP3_L_NOCP
; rung 46
LDNOT 10.04  ; CP3:GO
LD 10.09  ; CP3:L_CG
AND 10.05  ; CP3:L_NOCP
OR P_On  // 2015/11/13変更
ANDLD
ANDNOT 10.07  ; CP3:L_NCCP
OUT 622.02  ; CP3_L_NCCP
; rung 47
LDNOT 10.04  ; CP3:GO
LD 10.09  ; CP3:L_CG
AND 10.05  ; CP3:L_NOCP
AND 10.07  ; CP3:L_NCCP
OR P_On  // 2015/11/13変更
ANDLD
AND 10.11  ; CP3:L_未測定  // 2015/11/13変更
OUT 622.03  ; CP3_L_未測定
; rung 48
LDNOT 10.04  ; CP3:GO
ANDNOT 10.10  ; CP3:R_CG
LD 10.06  ; CP3:R_NOCP
OR P_On  // 2015/11/13変更
ANDLD
AND 10.08  ; CP3:R_NCCP
ANDNOT 622.07  ; CP3_R_NCCP
ANDNOT 622.10  ; CP3_L_NG
OUT 622.05  ; CP3_R_CG
; rung 49
LDNOT 10.04  ; CP3:GO
AND 10.10  ; CP3:R_CG
ANDNOT 10.06  ; CP3:R_NOCP
AND 10.08  ; CP3:R_NCCP
ANDNOT 622.05  ; CP3_R_CG
ANDNOT 622.07  ; CP3_R_NCCP
ANDNOT 622.10  ; CP3_L_NG
OUT 622.06  ; CP3_R_NOCP

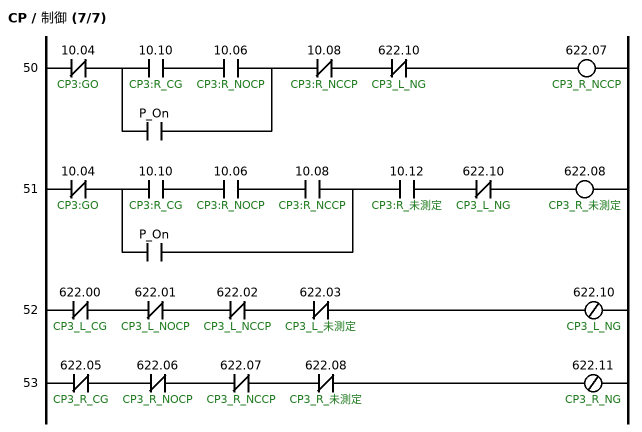
; rung 50
LDNOT 10.04  ; CP3:GO
LD 10.10  ; CP3:R_CG
AND 10.06  ; CP3:R_NOCP
OR P_On  // 2015/11/13変更
ANDLD
ANDNOT 10.08  ; CP3:R_NCCP
ANDNOT 622.10  ; CP3_L_NG
OUT 622.07  ; CP3_R_NCCP
; rung 51
LDNOT 10.04  ; CP3:GO
LD 10.10  ; CP3:R_CG
AND 10.06  ; CP3:R_NOCP
AND 10.08  ; CP3:R_NCCP
OR P_On  // 2015/11/13変更
ANDLD
AND 10.12  ; CP3:R_未測定  // 2015/11/13変更
ANDNOT 622.10  ; CP3_L_NG
OUT 622.08  ; CP3_R_未測定
; rung 52
LDNOT 622.00  ; CP3_L_CG
ANDNOT 622.01  ; CP3_L_NOCP
ANDNOT 622.02  ; CP3_L_NCCP
ANDNOT 622.03  ; CP3_L_未測定
OUTNOT 622.10  ; CP3_L_NG
; rung 53
LDNOT 622.05  ; CP3_R_CG
ANDNOT 622.06  ; CP3_R_NOCP
ANDNOT 622.07  ; CP3_R_NCCP
ANDNOT 622.08  ; CP3_R_未測定
OUTNOT 622.11  ; CP3_R_NG

### Section 出力

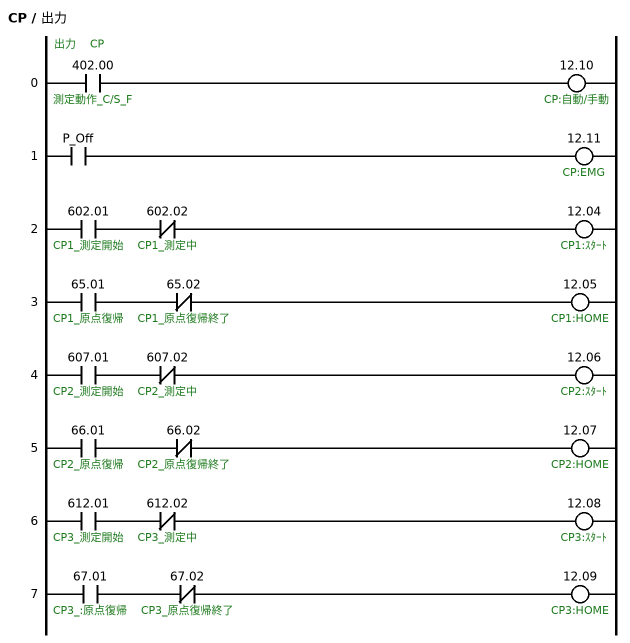
; rung 0: 出力    CP
LD 402.00  ; 測定動作_C/S_F
OUT 12.10  ; CP:自動/手動
; rung 1
LD P_Off
OUT 12.11  ; CP:EMG
; rung 2
LD 602.01  ; CP1_測定開始
ANDNOT 602.02  ; CP1_測定中
OUT 12.04  ; CP1:ｽﾀｰﾄ
; rung 3
LD 65.01  ; CP1_原点復帰
ANDNOT 65.02  ; CP1_原点復帰終了
OUT 12.05  ; CP1:HOME
; rung 4
LD 607.01  ; CP2_測定開始
ANDNOT 607.02  ; CP2_測定中
OUT 12.06  ; CP2:ｽﾀｰﾄ
; rung 5
LD 66.01  ; CP2_原点復帰
ANDNOT 66.02  ; CP2_原点復帰終了
OUT 12.07  ; CP2:HOME
; rung 6
LD 612.01  ; CP3_測定開始
ANDNOT 612.02  ; CP3_測定中
OUT 12.08  ; CP3:ｽﾀｰﾄ
; rung 7
LD 67.01  ; CP3_:原点復帰
ANDNOT 67.02  ; CP3_原点復帰終了
OUT 12.09  ; CP3:HOME

### Section ｴﾗｰ

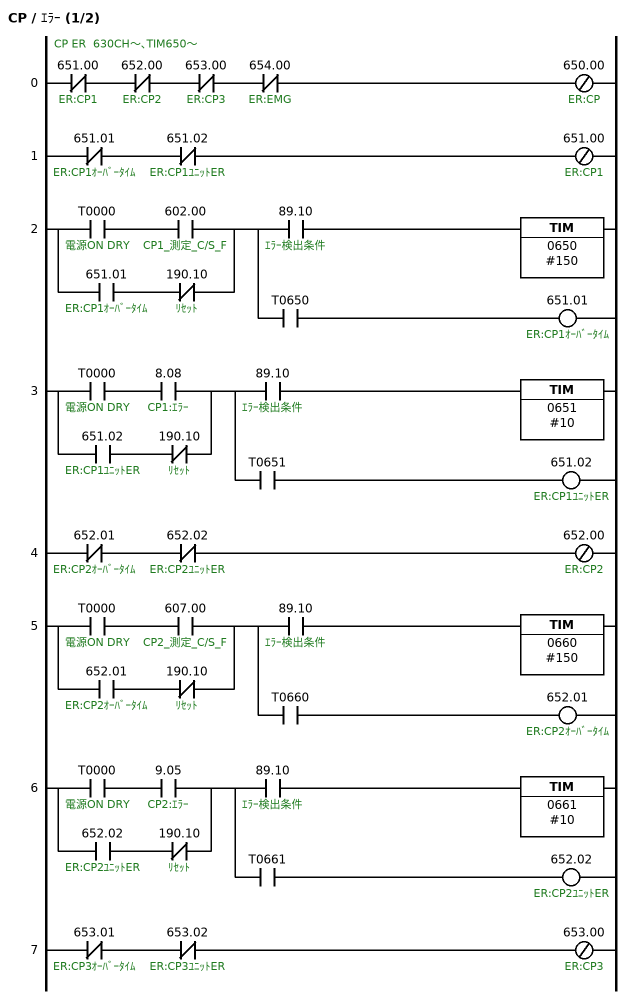
; rung 0: CP ER  630CH～､TIM650～
LDNOT 651.00  ; ER:CP1
ANDNOT 652.00  ; ER:CP2
ANDNOT 653.00  ; ER:CP3
ANDNOT 654.00  ; ER:EMG
OUTNOT 650.00  ; ER:CP
; rung 1
LDNOT 651.01  ; ER:CP1ｵｰﾊﾞｰﾀｲﾑ
ANDNOT 651.02  ; ER:CP1ﾕﾆｯﾄER
OUTNOT 651.00  ; ER:CP1
; rung 2
LD T0000  ; 電源ON DRY
AND 602.00  ; CP1_測定_C/S_F
LD 651.01  ; ER:CP1ｵｰﾊﾞｰﾀｲﾑ
ANDNOT 190.10  ; ﾘｾｯﾄ
ORLD
OUT TR0
AND 89.10  ; ｴﾗｰ検出条件
TIM 0650 #150
LD TR0
AND T0650
OUT 651.01  ; ER:CP1ｵｰﾊﾞｰﾀｲﾑ
; rung 3
LD T0000  ; 電源ON DRY
AND 8.08  ; CP1:ｴﾗｰ
LD 651.02  ; ER:CP1ﾕﾆｯﾄER
ANDNOT 190.10  ; ﾘｾｯﾄ
ORLD
OUT TR0
AND 89.10  ; ｴﾗｰ検出条件
TIM 0651 #10
LD TR0
AND T0651
OUT 651.02  ; ER:CP1ﾕﾆｯﾄER
; rung 4
LDNOT 652.01  ; ER:CP2ｵｰﾊﾞｰﾀｲﾑ
ANDNOT 652.02  ; ER:CP2ﾕﾆｯﾄER
OUTNOT 652.00  ; ER:CP2
; rung 5
LD T0000  ; 電源ON DRY
AND 607.00  ; CP2_測定_C/S_F
LD 652.01  ; ER:CP2ｵｰﾊﾞｰﾀｲﾑ
ANDNOT 190.10  ; ﾘｾｯﾄ
ORLD
OUT TR0
AND 89.10  ; ｴﾗｰ検出条件
TIM 0660 #150
LD TR0
AND T0660
OUT 652.01  ; ER:CP2ｵｰﾊﾞｰﾀｲﾑ
; rung 6
LD T0000  ; 電源ON DRY
AND 9.05  ; CP2:ｴﾗｰ
LD 652.02  ; ER:CP2ﾕﾆｯﾄER
ANDNOT 190.10  ; ﾘｾｯﾄ
ORLD
OUT TR0
AND 89.10  ; ｴﾗｰ検出条件
TIM 0661 #10
LD TR0
AND T0661
OUT 652.02  ; ER:CP2ﾕﾆｯﾄER
; rung 7
LDNOT 653.01  ; ER:CP3ｵｰﾊﾞｰﾀｲﾑ
ANDNOT 653.02  ; ER:CP3ﾕﾆｯﾄER
OUTNOT 653.00  ; ER:CP3

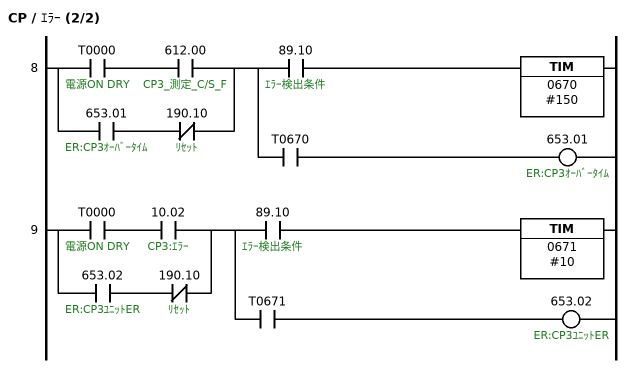
; rung 8
LD T0000  ; 電源ON DRY
AND 612.00  ; CP3_測定_C/S_F
LD 653.01  ; ER:CP3ｵｰﾊﾞｰﾀｲﾑ
ANDNOT 190.10  ; ﾘｾｯﾄ
ORLD
OUT TR0
AND 89.10  ; ｴﾗｰ検出条件
TIM 0670 #150
LD TR0
AND T0670
OUT 653.01  ; ER:CP3ｵｰﾊﾞｰﾀｲﾑ
; rung 9
LD T0000  ; 電源ON DRY
AND 10.02  ; CP3:ｴﾗｰ
LD 653.02  ; ER:CP3ﾕﾆｯﾄER
ANDNOT 190.10  ; ﾘｾｯﾄ
ORLD
OUT TR0
AND 89.10  ; ｴﾗｰ検出条件
TIM 0671 #10
LD TR0
AND T0671
OUT 653.02  ; ER:CP3ﾕﾆｯﾄER

### Section END
; rung 0
END(001)

## Program ﾃｰﾀ処理 (cyclic task 7)

### Section 判定保持

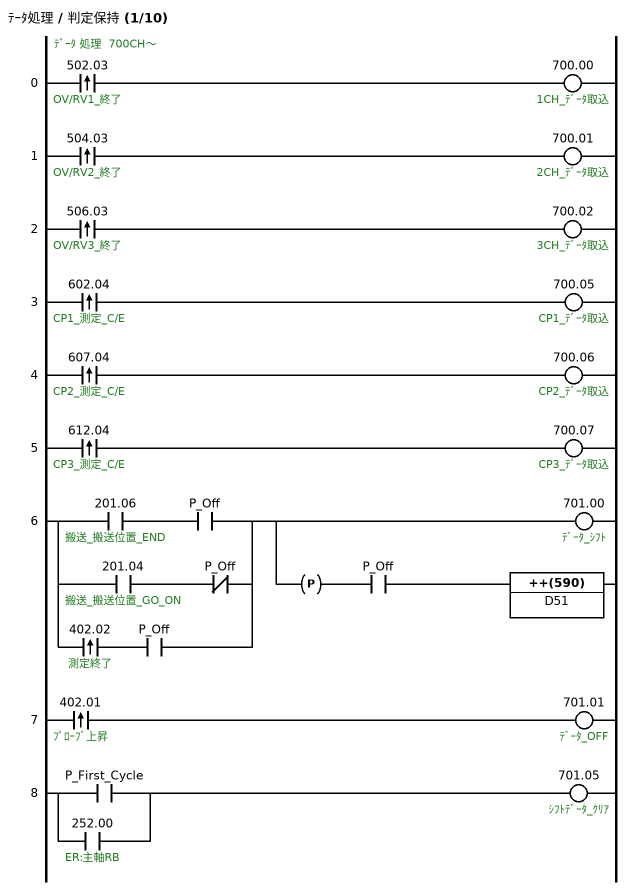
; rung 0: ﾃﾞｰﾀ 処理  700CH～
@LD 502.03  ; OV/RV1_終了
OUT 700.00  ; 1CH_ﾃﾞｰﾀ取込
; rung 1
@LD 504.03  ; OV/RV2_終了
OUT 700.01  ; 2CH_ﾃﾞｰﾀ取込
; rung 2
@LD 506.03  ; OV/RV3_終了
OUT 700.02  ; 3CH_ﾃﾞｰﾀ取込
; rung 3
@LD 602.04  ; CP1_測定_C/E
OUT 700.05  ; CP1_ﾃﾞｰﾀ取込
; rung 4
@LD 607.04  ; CP2_測定_C/E
OUT 700.06  ; CP2_ﾃﾞｰﾀ取込
; rung 5
@LD 612.04  ; CP3_測定_C/E
OUT 700.07  ; CP3_ﾃﾞｰﾀ取込
; rung 6
LD 201.06  ; 搬送_搬送位置_END
AND P_Off
LD 201.04  ; 搬送_搬送位置_GO_ON
ANDNOT P_Off
ORLD
@LD 402.02  ; 測定終了
AND P_Off
ORLD
OUT 701.00  ; ﾃﾞｰﾀ_ｼﾌﾄ
UP(521)
AND P_Off
++(590) D51
; rung 7
@LD 402.01  ; ﾌﾟﾛｰﾌﾞ上昇
OUT 701.01  ; ﾃﾞｰﾀ_OFF
; rung 8
LD P_First_Cycle
OR 252.00  ; ER:主軸RB
OUT 701.05  ; ｼﾌﾄﾃﾞｰﾀ_ｸﾘｱ

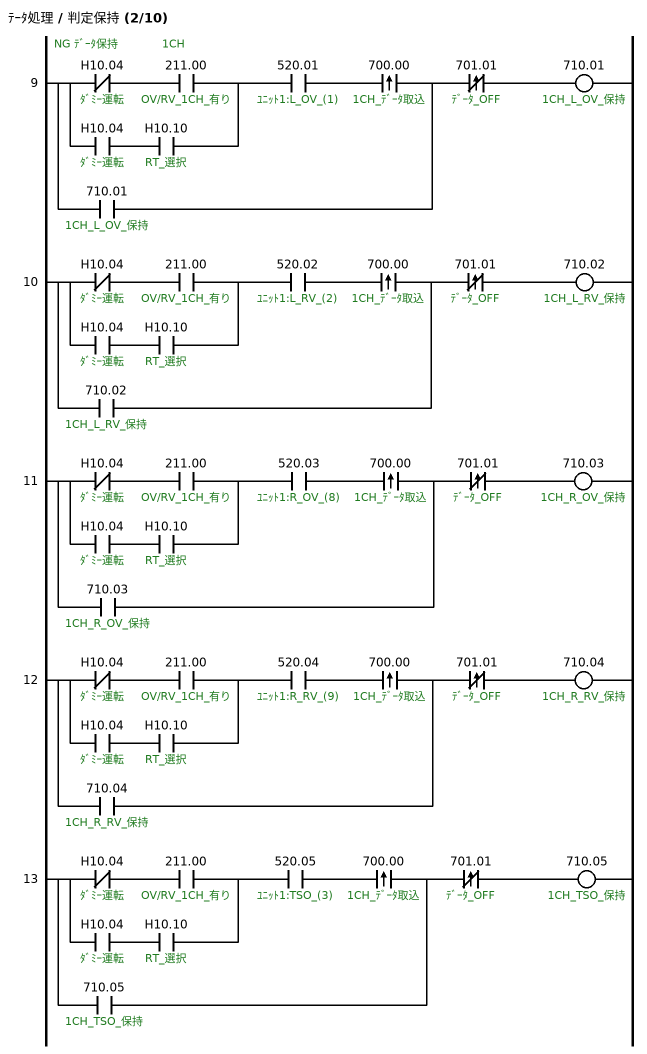
; rung 9: NG ﾃﾞｰﾀ保持　　　　1CH
LDNOT H10.04  ; ﾀﾞﾐｰ運転
AND 211.00  ; OV/RV_1CH_有り
LD H10.04  ; ﾀﾞﾐｰ運転
AND H10.10  ; RT_選択
ORLD
AND 520.01  ; ﾕﾆｯﾄ1:L_OV_(1)
@AND 700.00  ; 1CH_ﾃﾞｰﾀ取込
OR 710.01  ; 1CH_L_OV_保持
@ANDNOT 701.01  ; ﾃﾞｰﾀ_OFF
OUT 710.01  ; 1CH_L_OV_保持
; rung 10
LDNOT H10.04  ; ﾀﾞﾐｰ運転
AND 211.00  ; OV/RV_1CH_有り
LD H10.04  ; ﾀﾞﾐｰ運転
AND H10.10  ; RT_選択
ORLD
AND 520.02  ; ﾕﾆｯﾄ1:L_RV_(2)
@AND 700.00  ; 1CH_ﾃﾞｰﾀ取込
OR 710.02  ; 1CH_L_RV_保持
@ANDNOT 701.01  ; ﾃﾞｰﾀ_OFF
OUT 710.02  ; 1CH_L_RV_保持
; rung 11
LDNOT H10.04  ; ﾀﾞﾐｰ運転
AND 211.00  ; OV/RV_1CH_有り
LD H10.04  ; ﾀﾞﾐｰ運転
AND H10.10  ; RT_選択
ORLD
AND 520.03  ; ﾕﾆｯﾄ1:R_OV_(8)
@AND 700.00  ; 1CH_ﾃﾞｰﾀ取込
OR 710.03  ; 1CH_R_OV_保持
@ANDNOT 701.01  ; ﾃﾞｰﾀ_OFF
OUT 710.03  ; 1CH_R_OV_保持
; rung 12
LDNOT H10.04  ; ﾀﾞﾐｰ運転
AND 211.00  ; OV/RV_1CH_有り
LD H10.04  ; ﾀﾞﾐｰ運転
AND H10.10  ; RT_選択
ORLD
AND 520.04  ; ﾕﾆｯﾄ1:R_RV_(9)
@AND 700.00  ; 1CH_ﾃﾞｰﾀ取込
OR 710.04  ; 1CH_R_RV_保持
@ANDNOT 701.01  ; ﾃﾞｰﾀ_OFF
OUT 710.04  ; 1CH_R_RV_保持
; rung 13
LDNOT H10.04  ; ﾀﾞﾐｰ運転
AND 211.00  ; OV/RV_1CH_有り
LD H10.04  ; ﾀﾞﾐｰ運転
AND H10.10  ; RT_選択
ORLD
AND 520.05  ; ﾕﾆｯﾄ1:TSO_(3)
@AND 700.00  ; 1CH_ﾃﾞｰﾀ取込
OR 710.05  ; 1CH_TSO_保持
@ANDNOT 701.01  ; ﾃﾞｰﾀ_OFF
OUT 710.05  ; 1CH_TSO_保持

